// TIA Portal V19 export
ORGANIZATION_BLOCK "Main"   // OB2601, LAD, ProgramCycle
TITLE = "Main Program Sweep (Cycle)"
// stored: AutoNumber false, Namespace Unit2.Em5, SetENOAutomatically false
   VAR_INPUT
      Initial_Call : Bool;   // Initial call of this OB
      Remanence : Bool;   // =True, if remanent data are available
   END_VAR
BEGIN

REGION Network 1 (SCL)
   "Unit2.Em5.instSimulation"();

   "Unit2.Em5.CallEquipment_DB"(unitStatus:="Unit2.EmNodes".unitStatus,
                    unitAlarmDB:="Unit2.Alarms".emAlarms[Unit2_EM5],
                    emFeedback:="Unit2.EmNodes".emFeedback[Unit2_EM5]);
END_REGION
END_ORGANIZATION_BLOCK
